{attribute 'qualified_only'}
VAR_GLOBAL CONSTANT
	strExportDirectory : STRING := 'C:\TwinCAT\3.1\Boot\CurrentConfig\';
END_VAR

(* stored: Version 1.1.0.1
   GVL GVL_Parameter: Id {06b1eece-8629-4f9e-b6a4-2d2d8f628d63}, ParameterList True *)
